Universal Robots PolyScope program: 20250617_LR-upup.urp

Program 20250617_LR-upup (installation=20240827 directory=/programs/Demos/vision/test createdIn=5.13.1 lastSavedIn=5.15.1 robotSerialNumber=20245500285)
Calibrated DH parameters: a=[0.000097, -0.210459, -0.026602, 0.000137, 0.000078, 0]; d=[0.162601, 254.180657, -54.076236, -199.970743, 0.099615, 0.099684]; alpha=[1.569796, -0.001455, 0.001957, 1.570525, -1.571561, 0]; deltaTheta=[0, -1.053331, 8.839472, -1.50296, 0.000002, 0]
InitVariablesNode
Robot Program (runOnlyOnce=false)
  MoveJ speed 180 deg/s, acceleration 400 deg/s^2 (useActiveTCP=true positionType=JointAngles) feature=Base
    Waypoint 路点_1: TCP in base x=104.511 y=-367.887 z=150.56 mm, rx=-1.9493 ry=-1.8262 rz=-0.6048 rad; joints [85.471, -80.224, 100.082, -75.625, -90.165, 89.439] deg; TCP offset x=-0.17 y=0 z=192.95 mm, rx=0 ry=0 rz=0 rad
    If False
      Waypoint tttt: TCP in base x=121.665 y=-533.03 z=1.173 mm, rx=2.2461 ry=2.1952 rz=0.0012 rad; joints [88.581, -70.11, 113.379, -133.317, -90.004, 90.059] deg
  If True
    offs1 := [-0.18,-0.05]
    offs2 := [-0.18,0.05]
    offs3 := [-0.1,-0.05]
    offs4 := [-0.1,0.05]
    offs5 := [0.1,-0.05]
    offs6 := [0.1,0.05]
    offs7 := [0.18,-0.05]
    offs8 := [0.18,0.05]
  If True
    p1 := pose_add(tttt, p[offs1[0],offs1[1],0,0,0,0])
    p2 := pose_add(tttt, p[offs2[0],offs2[1],0,0,0,0])
    p3 := pose_add(tttt, p[offs3[0],offs3[1],0,0,0,0])
    p4 := pose_add(tttt, p[offs4[0],offs4[1],0,0,0,0])
    p5 := pose_add(tttt, p[offs5[0],offs5[1],0,0,0,0])
    p6 := pose_add(tttt, p[offs6[0],offs6[1],0,0,0,0])
    p7 := pose_add(tttt, p[offs7[0],offs7[1],0,0,0,0])
    p8 := pose_add(tttt, p[offs8[0],offs8[1],0,0,0,0])
  If True
    Script: vision = rpc_factory("xmlrpc","http://192.168.1.7:9121/RPC2")
    Script: gripper = rpc_factory("xmlrpc","http://192.168.1.7:9120/RPC2")
    Script: gripper.open()
  If True
    qqq := 0
    h_up := 0.1
    group1 := [p1,p2,p3,p4]
    group2 := [p5,p6,p7,p8]
  Loop Forever
    'g1'
    Loop While (checkContinuously=false) expression=qqq≤1
      n := 0
      qqq := 2
      MoveJ speed 180 deg/s, acceleration 400 deg/s^2 (useActiveTCP=true positionType=JointAngles) feature=Base
        Waypoint 路点_1: TCP in base x=104.511 y=-367.887 z=150.56 mm, rx=-1.9493 ry=-1.8262 rz=-0.6048 rad; joints [85.471, -80.224, 100.082, -75.625, -90.165, 89.439] deg
        Wait Sleep waitTime=0.5
      campose := get_actual_tcp_pose()
      take := True
      Loop While (checkContinuously=false) expression=take== True
        photo := vision.take_photo(campose)
        If photo≠ True
          Popup Message (haltProgram=false message=continues? inputType=Text)
        Else 
          take := False
      articlenum := vision.get_obj_num()
      Loop While (checkContinuously=false) expression=n<articlenum
        obj_num := n
        pose := p[0.0,0.0,0.0,2.221,2.221,0.004]
        obj_pose := vision.get_obj_pose(obj_num)
        Script: pose[0]=obj_pose[0]
        Script: pose[1]=obj_pose[1]
        Script: pose[2]=obj_pose[2]+0.025
        Script: pose[3]=obj_pose[3]
        Script: pose[4]=obj_pose[4]
        Script: pose[5]=obj_pose[5]
        MoveL speed 3000 mm/s, acceleration 6000 mm/s^2 (useActiveTCP=true) feature=Base
          Waypoint Variable (Variable): variable(name=pose)
        Script: pose[2]=obj_pose[2] - 0.06
        If pose[2]<0.003
          Script: pose[2] = 0.003
        MoveL speed 3000 mm/s, acceleration 6000 mm/s^2 (useActiveTCP=true) feature=Base
          Waypoint Variable (Variable): variable=pose
          Script: gripper.adaptiveClose()
        first_pose := pose
        Script: pose[2]=pose[2] + h_up
        MoveL speed 3000 mm/s, acceleration 6000 mm/s^2 (useActiveTCP=true) feature=Base
          Waypoint Variable (Variable): variable=pose
        target_pose := group1[n]
        Script: target_pose[2]=first_pose[2]
        down_pose := target_pose
        Script: down_pose[2]=down_pose[2] + h_up
        MoveL speed 3000 mm/s, acceleration 6000 mm/s^2 (useActiveTCP=true) feature=Base
          Waypoint Variable (Variable): variable=down_pose
        MoveL speed 3000 mm/s, acceleration 6000 mm/s^2 (useActiveTCP=true) feature=Base
          Waypoint Variable (Variable): variable(name=target_pose)
          Script: gripper.open()
        MoveL speed 3000 mm/s, acceleration 6000 mm/s^2 (useActiveTCP=true) feature=Base
          Waypoint Variable (Variable): variable=down_pose
        n := n + 1
    'g2'
    Loop While (checkContinuously=false) expression=qqq≥2
      n := 0
      qqq := 1
      MoveJ speed 180 deg/s, acceleration 400 deg/s^2 (useActiveTCP=true positionType=JointAngles) feature=Base
        Waypoint 路点_1: TCP in base x=104.511 y=-367.887 z=150.56 mm, rx=-1.9493 ry=-1.8262 rz=-0.6048 rad; joints [85.471, -80.224, 100.082, -75.625, -90.165, 89.439] deg
        Wait Sleep waitTime=0.5
      campose := get_actual_tcp_pose()
      take := True
      Loop While (checkContinuously=false) expression=take== True
        photo := vision.take_photo(campose)
        If photo≠ True
          Popup Message (haltProgram=false message=continues? inputType=Text)
        Else 
          take := False
      articlenum := vision.get_obj_num()
      Loop While (checkContinuously=false) expression=n<articlenum
        obj_num := n
        pose := p[0.0,0.0,0.0,2.221,2.221,0.004]
        obj_pose := vision.get_obj_pose(obj_num)
        Script: pose[0]=obj_pose[0]
        Script: pose[1]=obj_pose[1]
        Script: pose[2]=obj_pose[2]+0.025
        Script: pose[3]=obj_pose[3]
        Script: pose[4]=obj_pose[4]
        Script: pose[5]=obj_pose[5]
        MoveL speed 3000 mm/s, acceleration 6000 mm/s^2 (useActiveTCP=true) feature=Base
          Waypoint Variable (Variable): variable=pose
        Script: pose[2]=obj_pose[2] - 0.06
        If pose[2]<0.003
          Script: pose[2] = 0.003
        MoveL speed 3000 mm/s, acceleration 6000 mm/s^2 (useActiveTCP=true) feature=Base
          Waypoint Variable (Variable): variable=pose
          Script: gripper.adaptiveClose()
        first_pose := pose
        Script: pose[2]=pose[2] + h_up
        MoveL speed 3000 mm/s, acceleration 6000 mm/s^2 (useActiveTCP=true) feature=Base
          Waypoint Variable (Variable): variable=pose
        target_pose := group2[n]
        Script: target_pose[2]=first_pose[2]
        down_pose := target_pose
        Script: down_pose[2]=down_pose[2] + h_up
        MoveL speed 3000 mm/s, acceleration 6000 mm/s^2 (useActiveTCP=true) feature=Base
          Waypoint Variable (Variable): variable=down_pose
        MoveL speed 3000 mm/s, acceleration 6000 mm/s^2 (useActiveTCP=true) feature=Base
          Waypoint Variable (Variable): variable=target_pose
          Script: gripper.open()
        MoveL speed 3000 mm/s, acceleration 6000 mm/s^2 (useActiveTCP=true) feature=Base
          Waypoint Variable (Variable): variable=down_pose
        n := n + 1
